// TIA Portal V19 export
FUNCTION "MODE SELECTION" : Void   // FC2, LAD
{ S7_Optimized_Access := 'TRUE' }
// stored: SetENOAutomatically false
   VAR_TEMP   // added for the SCL form of the ladder/FBD networks
      _w1 : Bool;
   END_VAR
BEGIN

REGION Network 1: STANDBY
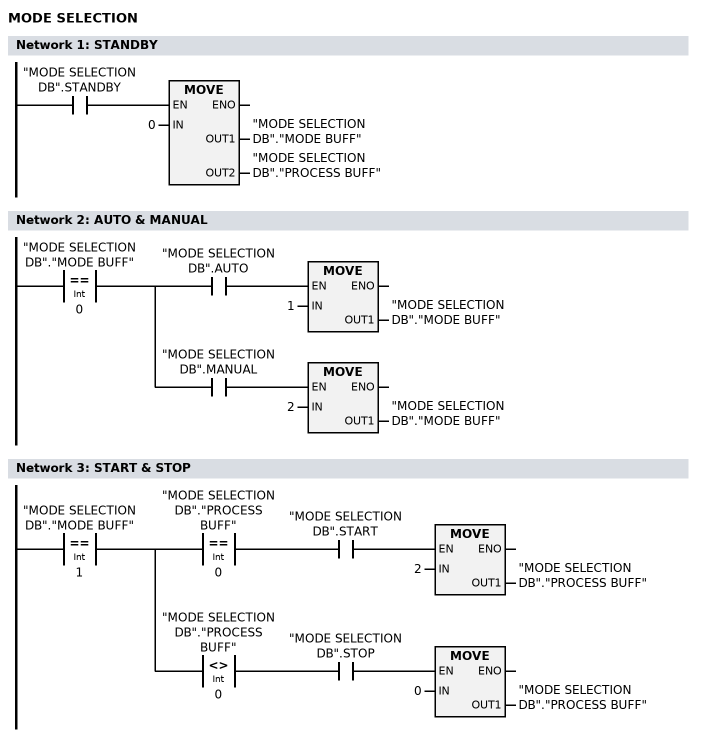
   RUNG wire#powerrail
      Contact( "MODE SELECTION DB".STANDBY )
      Move(in := 0, out1 => "MODE SELECTION DB"."MODE BUFF", out2 => "MODE SELECTION DB"."PROCESS BUFF")
   END_RUNG
   // the same network as SCL:
   IF "MODE SELECTION DB".STANDBY THEN
       "MODE SELECTION DB"."MODE BUFF" := 0;
       "MODE SELECTION DB"."PROCESS BUFF" := 0;
   END_IF;
END_REGION

REGION Network 2: AUTO & MANUAL
   RUNG wire#powerrail
      { S7_Templates := "SrcType := Int" } EQ_Contact(in1 := "MODE SELECTION DB"."MODE BUFF", in2 := 0)
      wire#w1
      Contact( "MODE SELECTION DB".AUTO )
      Move(in := 1, out1 => "MODE SELECTION DB"."MODE BUFF")
   END_RUNG
   RUNG wire#w1
      Contact( "MODE SELECTION DB".MANUAL )
      Move(in := 2, out1 => "MODE SELECTION DB"."MODE BUFF")
   END_RUNG
   // the same network as SCL:
   #_w1 := "MODE SELECTION DB"."MODE BUFF" = 0;
   IF #_w1 AND "MODE SELECTION DB".AUTO THEN "MODE SELECTION DB"."MODE BUFF" := 1; END_IF;
   IF #_w1 AND "MODE SELECTION DB".MANUAL THEN "MODE SELECTION DB"."MODE BUFF" := 2; END_IF;
END_REGION

REGION Network 3: START & STOP
   RUNG wire#powerrail
      { S7_Templates := "SrcType := Int" } EQ_Contact(in1 := "MODE SELECTION DB"."MODE BUFF", in2 := 1)
      wire#w1
      { S7_Templates := "SrcType := Int" } EQ_Contact(in1 := "MODE SELECTION DB"."PROCESS BUFF", in2 := 0)
      Contact( "MODE SELECTION DB".START )
      Move(in := 2, out1 => "MODE SELECTION DB"."PROCESS BUFF")
   END_RUNG
   RUNG wire#w1
      { S7_Templates := "SrcType := Int" } NE_Contact(in1 := "MODE SELECTION DB"."PROCESS BUFF", in2 := 0)
      Contact( "MODE SELECTION DB".STOP )
      Move(in := 0, out1 => "MODE SELECTION DB"."PROCESS BUFF")
   END_RUNG
   // the same network as SCL:
   #_w1 := "MODE SELECTION DB"."MODE BUFF" = 1;
   IF #_w1 AND ("MODE SELECTION DB"."PROCESS BUFF" = 0) AND "MODE SELECTION DB".START THEN
       "MODE SELECTION DB"."PROCESS BUFF" := 2;
   END_IF;
   IF #_w1 AND ("MODE SELECTION DB"."PROCESS BUFF" <> 0) AND "MODE SELECTION DB".STOP THEN
       "MODE SELECTION DB"."PROCESS BUFF" := 0;
   END_IF;
END_REGION
END_FUNCTION
